TYPE ST_PlcEventHmi :
STRUCT
	nEventID:INT;
	nEventType:INT;	(*1:Alarm , 2:Warning , *)
	nEventColor:UDINT;
	nTextColor:UDINT;
	sEventTime:STRING(32);
	sEventAckTime:STRING(32);
END_STRUCT
END_TYPE

(* stored: Version 1.1.0.1, ProductVersion 3.1.4024.12
   DUT ST_PlcEventHmi: Id {c563a2e3-1509-4c3f-acb4-f78985702eaf} *)
